(* IEC 61131-3 sources: CS_4_Aufzugsteuerung/src/Stations/CP112/Steuerung/Class/clsEtagenSensorik, 1 file *)

(* ---- clsEtagenSensorik.st ---- *)
(*!
<Class
	Name               = "clsEtagenSensorik"
	Revision           = "0.0"
	RealtimeTask       = "false"
	CyclicTask         = "true"
	DefCyclictime      = "1 ms"
	BackgroundTask     = "false"
	Sigmatek           = "false"
	OSInterface        = "false"
	HighPriority       = "false"
	Automatic          = "false"
	UpdateMode         = "Prescan"
	SharedCommandTable = "true"
	Objectsize         = "(284,120)">
	<Channels>
		<Server Name="ClassSvr" Visualized="false" Initialize="false" WriteProtected="true" Retentive="false"/>
		<Server Name="sVisuEtage" Visualized="true" Initialize="false" WriteProtected="false" Retentive="false"/>
		<Client Name="cFahrzeit" Required="false" Internal="false"/>
		<Client Name="cStockwerke" Required="false" Internal="false"/>
		<Client Name="cTimer" Required="true" Internal="false"/>
	</Channels>
</Class>
*)
clsEtagenSensorik : CLASS
  //Servers:
	ClassSvr 	: SvrChCmd_DINT;
	sVisuEtage 	: SvrCh_DINT;
  //Clients:
	cTimer 	: CltChCmd_clsTimer;
	cFahrzeit 	: CltCh_UDINT;
	cStockwerke 	: CltCh_DINT;
  //Variables:
		xErreicht 	: BOOL;
		iEtage 	: DINT;
  //Functions:

	FUNCTION VIRTUAL GLOBAL CyWork
		VAR_INPUT
			EAX 	: UDINT;
		END_VAR
		VAR_OUTPUT
			state (EAX) 	: UDINT;
		END_VAR;

	FUNCTION GLOBAL hoch;

	FUNCTION GLOBAL runter;

	FUNCTION GLOBAL AktEtage
		VAR_OUTPUT
			iOut 	: DINT;
		END_VAR;

	FUNCTION GLOBAL erreicht
		VAR_OUTPUT
			xOut 	: BOOL;
		END_VAR;
  //Tables:
	FUNCTION @STD
		VAR_OUTPUT
			ret_code	: CONFSTATES;
		END_VAR;
	FUNCTION GLOBAL TAB @CT_;
END_CLASS;

#pragma usingLtd clsTimer

FUNCTION VIRTUAL GLOBAL clsEtagenSensorik::CyWork
	VAR_INPUT
		EAX 	: UDINT;
	END_VAR
	VAR_OUTPUT
		state (EAX) 	: UDINT;
	END_VAR

  // client einlesen
  cFahrzeit := cFahrzeit.Read();
  cStockwerke := cStockwerke.Read();

  //Uebergabe an HMI
  sVisuEtage := iEtage;

	state := READY;

END_FUNCTION

FUNCTION GLOBAL clsEtagenSensorik::hoch

// Init
xErreicht := FALSE;

// Prüfen ob bereits in der obersten Etage
IF iEtage >= cStockwerke THEN
    xErreicht := TRUE;
ELSE
    IF NOT cTimer.running() THEN
        cTimer.Start(_time := cFahrzeit);
    END_IF;

    // Fahrzeit abgelaufen
    IF cTimer.elapsed() THEN
        iEtage := iEtage + 1;
        xErreicht := TRUE;
        cTimer.reset();
    END_IF;
END_IF;

END_FUNCTION

FUNCTION GLOBAL clsEtagenSensorik::runter

// Init
xErreicht := FALSE;

// Prüfen ob bereits in der untersten Etage
IF iEtage <= 0 THEN
    xErreicht := TRUE;
ELSE
    IF NOT cTimer.running() THEN
        cTimer.Start(_time := cFahrzeit);
    END_IF;

    // Fahrzeit abgelaufen
    IF cTimer.elapsed() THEN
        iEtage := iEtage - 1;
        xErreicht := TRUE;
        cTimer.reset();
    END_IF;
END_IF;

END_FUNCTION

FUNCTION GLOBAL clsEtagenSensorik::AktEtage
	VAR_OUTPUT
		iOut 	: DINT;
	END_VAR
iOut := iEtage; //Noch unklar ob und wie iEtage bei Steuerung aufstart initialisiert wird

END_FUNCTION

FUNCTION GLOBAL clsEtagenSensorik::erreicht
	VAR_OUTPUT
		xOut 	: BOOL;
	END_VAR
 xOut := xErreicht;
END_FUNCTION
